{attribute 'qualified_only'}
{attribute 'strict'}
{attribute 'to_string'}
{info 'E_APP_VARIANT placeholder for application variant; add new members here'}
TYPE E_APP_VARIANT :
(
  VARIANT_INVALID
);
END_TYPE

(* stored: Version 1.1.0.1
   DUT E_APP_VARIANT: Id {a010c5da-5f20-4d7f-8bf2-caf9a44f9ab9} *)
